FUNCTION_BLOCK DeserializerParent
VAR
	children : List;
END_VAR

METHOD PUBLIC DeregisterChild
VAR_INPUT
	Child : I_Deserializer;
END_VAR
children.TryRemoveItem(Child);
END_METHOD

METHOD PUBLIC RegisterChild
VAR_INPUT
	Child : I_Deserializer;
END_VAR
children.AddItem(Child);
END_METHOD

END_FUNCTION_BLOCK

(* stored: Version 1.1.0.1, ProductVersion 3.1.4024.12
   POU DeserializerParent: Id {56b440c7-8c49-40a5-9bf4-bcd28d963269}, SpecialFunc None
   Method DeregisterChild: Id {a9622af3-00a7-433b-80e5-6cc2c1e9431c}
   Method RegisterChild: Id {a0da1f75-d2a3-4ca9-9272-73a1643dd9f8} *)
